{attribute addProperty BoxType "EL3443-0000-0016"}
{attribute addProperty Id "Voltage_Last_Zero_CrossingAT %I*ULINT648"}
{attribute addProperty CRC "1102320901"}
{attribute addProperty SizeInBites "64"}
{attribute addProperty SizeInBytes "8"}
TYPE L2_Timing_41B41505 :
STRUCT
	{attribute addProperty Name "Voltage_Last_Zero_Crossing"}
	Voltage_Last_Zero_Crossing AT %I* : ULINT;
END_STRUCT
END_TYPE

(* stored: Version 1.2.0.0, ProductVersion 3.1.4024.9
   DUT L2_Timing_41B41505: Id {3958976b-ca4f-4686-8e2e-7e59c9923195} *)
